(* LS Electric XG5000 project: XMC_MultiAxis_FBs *)
(* sample programs for multi-axis function blocks. *)
(* PLC LSPLC *)
(* module base 0 slot 0: Input/Output Module:XMC-DN24 (DC 24V Input 8Points/TR output 16Points) *)
(* module base 0 slot 1: Internal Analog Input/Output:XMF-AH04E (A/D voltage/current 2 channels, D/A voltage 2 channels) *)
(* task Periodic Task: Kind=2 *)
(* task Initialization Task: Kind=1 *)
(* task NC Program: Kind=6 *)

PROGRAM ECAT_Connect_Example (* task: Scan Program *)
VAR
    Connect_Error : BOOL; (* status that LS_Connect has an error *)
    Connect_ErrorID : WORD; (* LS_Connect Error number *)
    Connect_INST : LS_CONNECT; (* LS_Connect fb *)
    Disconnect_Error : BOOL; (* status that LS_Disconnect has an error *)
    Disconnect_ErrorID : WORD; (* Error Number for LS_Disconnect FB *)
    Disconnect_INST : LS_DISCONNECT; (* LS_Disconnect fb *)
    Execute_Connect : BOOL; (* Execute LS_Connect fb *)
    Execute_Disconnect : BOOL; (* execute LS_Disconnect fb *)
END_VAR

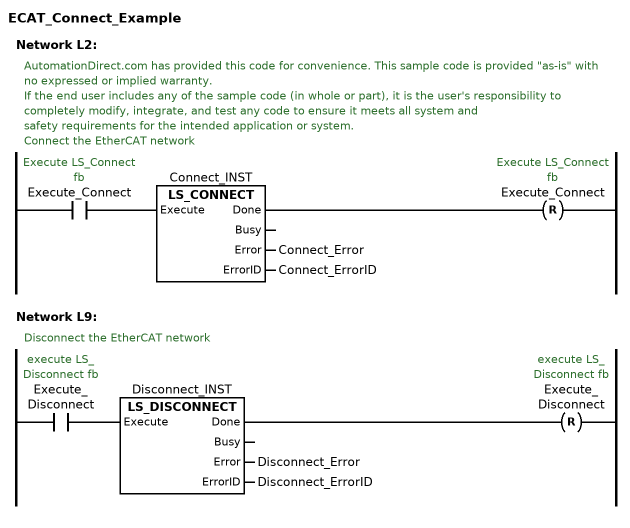
(* AutomationDirect.com has provided this code for convenience. This sample code is provided "as-is" with no expressed or implied warranty. / If the end user includes any of the sample code (in whole or part), it is the user's responsibility to completely modify, integrate, and test any code to ensure it meets all system and / safety requirements for the intended application or system. *)
(* Connect the EtherCAT network *)
(* Rung L2 *)
Connect_INST(Execute := Execute_Connect, Error => Connect_Error, ErrorID => Connect_ErrorID);
IF Connect_INST.Done THEN Execute_Connect := FALSE; END_IF;
(* Disconnect the EtherCAT network *)
(* Rung L9 *)
Disconnect_INST(Execute := Execute_Disconnect, Error => Disconnect_Error, ErrorID => Disconnect_ErrorID);
IF Disconnect_INST.Done THEN Execute_Disconnect := FALSE; END_IF;
END_PROGRAM

PROGRAM MC_PowerAll_Example (* task: Scan Program *)
(* example program for MC_PowerAll *)
VAR
    All_Axes_Ready : BOOL; (* flag that all axes are ready *)
    PowerAll_Error : BOOL; (* status of MC_Power error status *)
    PowerAll_ErrorID : WORD; (* error id of Axis 1 MC_Power *)
    PowerAll_INST : MC_POWERALL; (* MC_PowerALL fb *)
    PowerAll_Status : BOOL; (* status of axis 1 power *)
    PowerAll_Valid : BOOL; (* Axis1 power status is valid *)
    Power_On_Axis1 : BOOL; (* command to turn on power to axis 1 *)
END_VAR

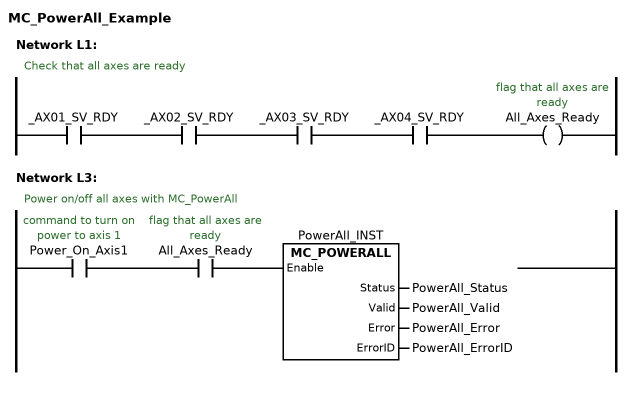
(* Check that all axes are ready *)
(* Rung L1 *)
All_Axes_Ready := _AX01_SV_RDY AND _AX02_SV_RDY AND _AX03_SV_RDY AND _AX04_SV_RDY;
(* Power on/off all axes with MC_PowerAll *)
(* Rung L3 *)
PowerAll_INST(Enable := Power_On_Axis1 AND All_Axes_Ready, Status => PowerAll_Status, Valid => PowerAll_Valid, Error => PowerAll_Error, ErrorID => PowerAll_ErrorID);
END_PROGRAM

PROGRAM Home_Example (* task: Scan Program *)
(* example of MC_Home and LS_Home *)
VAR
    All_Axes_Pwr_On : BOOL; (* status that all axes are powered on *)
    All_Axes_Ready : BOOL; (* flag that all axes are ready *)
    Execute_LS_HomeAll : BOOL; (* Execute LS_Home fb *)
    Execute_MC_HomeAll : BOOL; (* execute MC_Home fb *)
    LSHomeAll_Aborted : BOOL; (* LS_Home fb command aborted status *)
    LSHomeAll_Active : BOOL; (* LS_Home fb active status *)
    LSHomeAll_Busy : BOOL; (* LS_Home busy status *)
    LSHomeAll_Error : BOOL; (* LSHome fb error status *)
    LSHomeAll_ErrorID : WORD; (* LS_Home fb error id value *)
    LSHomeAll_INST : LS_HOMEALL; (* LS_HomeAll fb *)
    MCHomeAll_Aborted : BOOL; (* MC_Home command was aborted *)
    MCHomeAll_Active : BOOL; (* MC_Home is active *)
    MCHomeAll_Busy : BOOL; (* MC_Home is busy *)
    MCHomeAll_Error : BOOL; (* error status of MC_Home *)
    MCHomeAll_ErrorID : WORD; (* error id value for MC_Home *)
    MCHomeAll_INST : MC_HOMEALL; (* MC_HomeAll fb *)
END_VAR

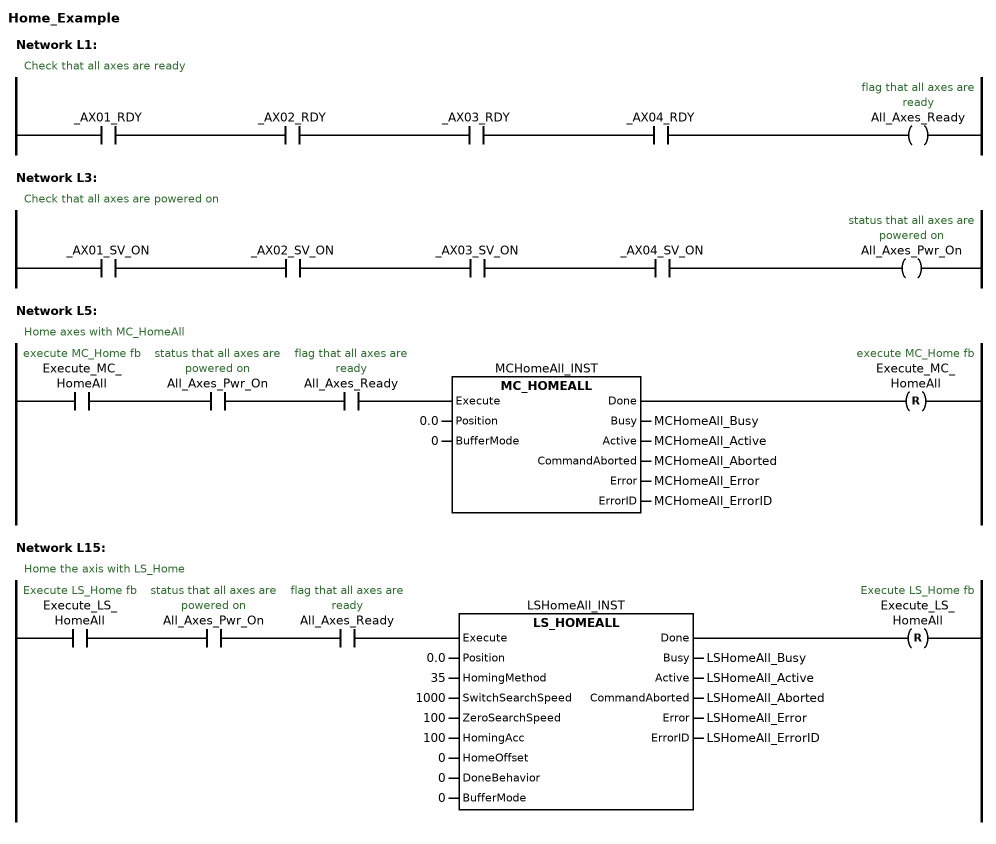
(* Check that all axes are ready *)
(* Rung L1 *)
All_Axes_Ready := _AX01_RDY AND _AX02_RDY AND _AX03_RDY AND _AX04_RDY;
(* Check that all axes are powered on *)
(* Rung L3 *)
All_Axes_Pwr_On := _AX01_SV_ON AND _AX02_SV_ON AND _AX03_SV_ON AND _AX04_SV_ON;
(* Home axes with MC_HomeAll *)
(* Rung L5 *)
MCHomeAll_INST(Execute := Execute_MC_HomeAll AND All_Axes_Pwr_On AND All_Axes_Ready, Position := 0.0, BufferMode := 0, Busy => MCHomeAll_Busy, Active => MCHomeAll_Active, CommandAborted => MCHomeAll_Aborted, Error => MCHomeAll_Error, ErrorID => MCHomeAll_ErrorID);
IF MCHomeAll_INST.Done THEN Execute_MC_HomeAll := FALSE; END_IF;
(* Home the axis with LS_Home *)
(* Rung L15 *)
LSHomeAll_INST(Execute := Execute_LS_HomeAll AND All_Axes_Pwr_On AND All_Axes_Ready, Position := 0.0, HomingMethod := 35, SwitchSearchSpeed := 1000, ZeroSearchSpeed := 100, HomingAcc := 100, HomeOffset := 0, DoneBehavior := 0, BufferMode := 0, Busy => LSHomeAll_Busy, Active => LSHomeAll_Active, CommandAborted => LSHomeAll_Aborted, Error => LSHomeAll_Error, ErrorID => LSHomeAll_ErrorID);
IF LSHomeAll_INST.Done THEN Execute_LS_HomeAll := FALSE; END_IF;
END_PROGRAM

PROGRAM MCStopAll_MCHaltAll_Examples (* task: Scan Program *)
(* Examples of MC_Stop and MC_Hault function blocks. *)
VAR
    All_Axes_Pwr_On : BOOL; (* status that all axes are powered on *)
    All_Axes_Ready : BOOL; (* flag that all axes are ready *)
    Execute_MCHaltAll : BOOL; (* execute MC_Halt FB *)
    Execute_MCStopAll : BOOL; (* command to execute MC_Stop fb *)
    MCHaltAll_Aborted : BOOL; (* MC_Hault command aborted status *)
    MCHaltAll_Active : BOOL; (* MC_Halt active status *)
    MCHaltAll_Busy : BOOL; (* Busy status for MC_Halt *)
    MCHaltAll_Error : BOOL; (* MC_Halt error status *)
    MCHaltAll_ErrorID : WORD; (* MC_Halt Error identification value *)
    MCHaltAll_INST : MC_HALTALL; (* MC_HaltAll fb *)
    MCStopAll_Aborted : BOOL; (* MC_Stop aborted status *)
    MCStopAll_Busy : BOOL; (* MC_Stop Busy Status *)
    MCStopAll_Error : BOOL; (* MC_Stop error status *)
    MCStopAll_ErrorID : WORD; (* MC_Stop error identification value *)
    MCStopAll_INST : MC_STOPALL; (* MC_Stop function block *)
END_VAR

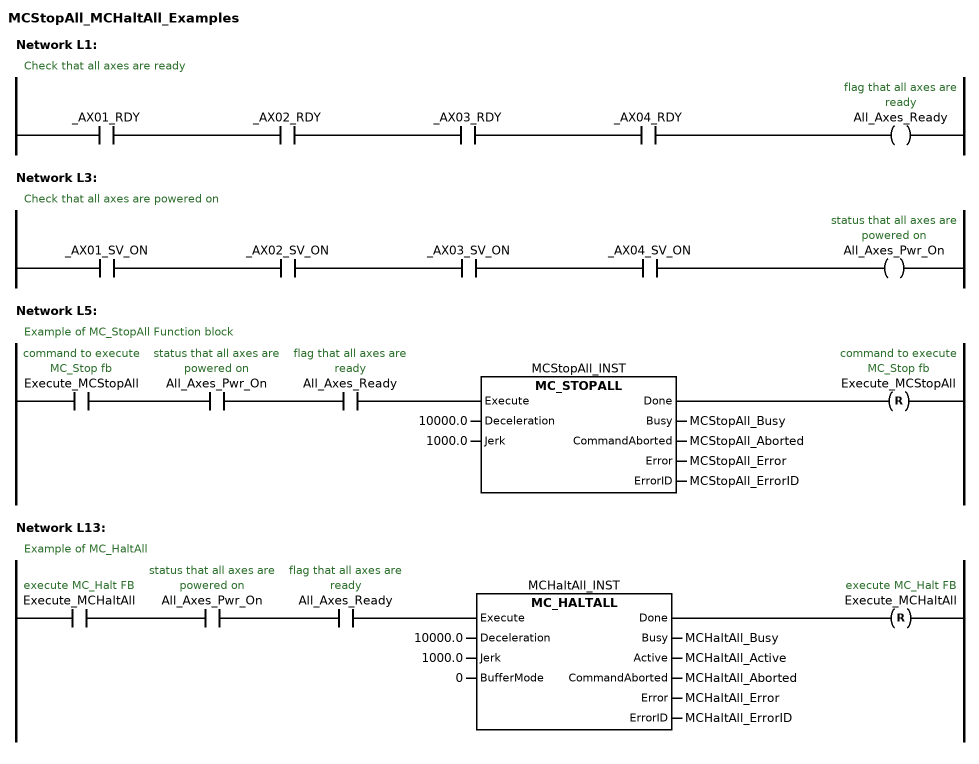
(* Check that all axes are ready *)
(* Rung L1 *)
All_Axes_Ready := _AX01_RDY AND _AX02_RDY AND _AX03_RDY AND _AX04_RDY;
(* Check that all axes are powered on *)
(* Rung L3 *)
All_Axes_Pwr_On := _AX01_SV_ON AND _AX02_SV_ON AND _AX03_SV_ON AND _AX04_SV_ON;
(* Example of MC_StopAll Function block *)
(* Rung L5 *)
MCStopAll_INST(Execute := Execute_MCStopAll AND All_Axes_Pwr_On AND All_Axes_Ready, Deceleration := 10000.0, Jerk := 1000.0, Busy => MCStopAll_Busy, CommandAborted => MCStopAll_Aborted, Error => MCStopAll_Error, ErrorID => MCStopAll_ErrorID);
IF MCStopAll_INST.Done THEN Execute_MCStopAll := FALSE; END_IF;
(* Example of MC_HaltAll *)
(* Rung L13 *)
MCHaltAll_INST(Execute := Execute_MCHaltAll AND All_Axes_Pwr_On AND All_Axes_Ready, Deceleration := 10000.0, Jerk := 1000.0, BufferMode := 0, Busy => MCHaltAll_Busy, Active => MCHaltAll_Active, CommandAborted => MCHaltAll_Aborted, Error => MCHaltAll_Error, ErrorID => MCHaltAll_ErrorID);
IF MCHaltAll_INST.Done THEN Execute_MCHaltAll := FALSE; END_IF;
END_PROGRAM

PROGRAM MC_Reset2All_Example (* task: Scan Program *)
(* example of MC_Reset2All function block. *)
VAR
    All_Axes_Ready : BOOL; (* flag that all axes are ready *)
    Execute_MCReset2All : BOOL; (* command to execute MC_Reset2 *)
    Reset2All_Busy : BOOL; (* busy status for MC_Reset2 *)
    Reset2All_Error : BOOL; (* error status for MC_Reset2 *)
    Reset2All_ErrorID : WORD; (* MC_Reset2 error identification *)
    Reset2All_ErrorType : UINT; (* error type for MC_Reset2 *)
    Reset2All_INST : MC_RESET2ALL; (* MC_Reset2All fb *)
END_VAR

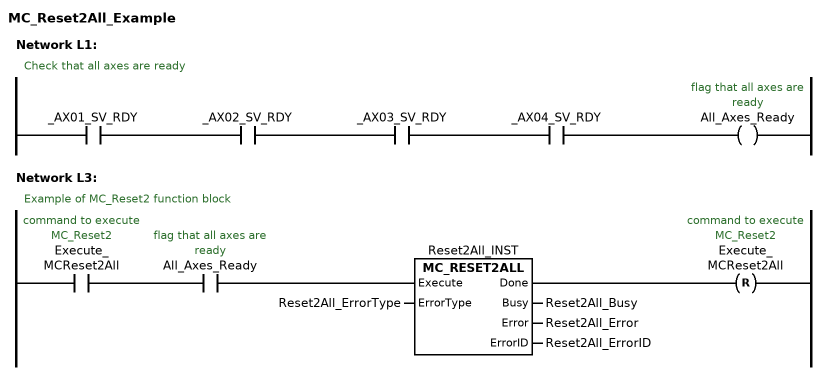
(* Check that all axes are ready *)
(* Rung L1 *)
All_Axes_Ready := _AX01_SV_RDY AND _AX02_SV_RDY AND _AX03_SV_RDY AND _AX04_SV_RDY;
(* Example of MC_Reset2 function block *)
(* Rung L3 *)
Reset2All_INST(Execute := Execute_MCReset2All AND All_Axes_Ready, ErrorType := Reset2All_ErrorType, Busy => Reset2All_Busy, Error => Reset2All_Error, ErrorID => Reset2All_ErrorID);
IF Reset2All_INST.Done THEN Execute_MCReset2All := FALSE; END_IF;
END_PROGRAM

PROGRAM MC_CamIn_CamOut_Example (* task: Scan Program *)
(* Example of MC_CamIn and MC_CamOut function block *)
VAR
    All_Axes_Pwr_On : BOOL; (* status that all axes are powered on *)
    All_Axes_Ready : BOOL; (* flag that all axes are ready *)
    CamIn_Aborted : BOOL; (* MC_CamIn command aborted status *)
    CamIn_Active : BOOL; (* MC_CamIn active status *)
    CamIn_Busy : BOOL; (* MC_CamIn busy status *)
    CamIn_CamTableID : UINT; (* Cam profle table id for MC_CamIn *)
    CamIn_ContinuousUpdate : BOOL; (* Continuous update input of MC_CamIn *)
    CamIn_EndOfProfile : BOOL; (* MC_CamIn end of profile status *)
    CamIn_Error : BOOL; (* MC_CamIn error status *)
    CamIn_ErrorID : WORD; (* MC_CamIn error identification *)
    CamIn_INST : MC_CAMIN; (* MC_CamIn fb *)
    CamIn_MasterOffset : LREAL; (* Master offset of MC_CamIn *)
    CamIn_MasterScaling : LREAL; (* Master scaling for MC_CamIn *)
    CamIn_MasterStartDistance : LREAL; (* Master Start distance for MC_CamIn *)
    CamIn_MasterSyncPosition : LREAL; (* Master Sync Position for MC_CamIn *)
    CamIn_MasterValueSource : UINT; (* Master value source for MC_CamIn *)
    CamIn_SlaveOffset : LREAL; (* Slave offset of MC_CamIn *)
    CamIn_SlaveScaling : LREAL; (* slave scaling MC_CamIn *)
    CamIn_StartMode : UINT; (* Start mode for MC_CamIn *)
    CamOut_Busy : BOOL; (* MC_CamOut busy status *)
    CamOut_Error : BOOL; (* error status for MC_CamOut *)
    CamOut_ErrorID : WORD; (* Error identification for MC_CamOut *)
    CamOut_INST : MC_CAMOUT; (* MC_CamOut function block *)
    Execute_CamIn : BOOL; (* execute MC_CamIn *)
    Execute_CamOut : BOOL; (* execute MC_CamOut function block *)
    Execute_MoveVelocity : BOOL; (* execute the MC_MoveVelocity Function block *)
    Master_Axis : UINT; (* master axis of MC_CamIn *)
    Slave_Axis : UINT; (* slave axis of MC_CamIn *)
    VelocityMove_Aborted : BOOL; (* MC_MoveVelocity Status aborted *)
    VelocityMove_Active : BOOL; (* active status of MC_MoveVelocity *)
    VelocityMove_Busy : BOOL; (* busy status of MC_MoveVelocity *)
    VelocityMove_Error : BOOL; (* Error status of MC_MoveVelocity *)
    VelocityMove_ErrorID : WORD; (* MC_MoveVelocity error identification *)
    Velocity_INST : MC_MOVEVELOCITY; (* MC_MoveVelocity function block instance *)
END_VAR

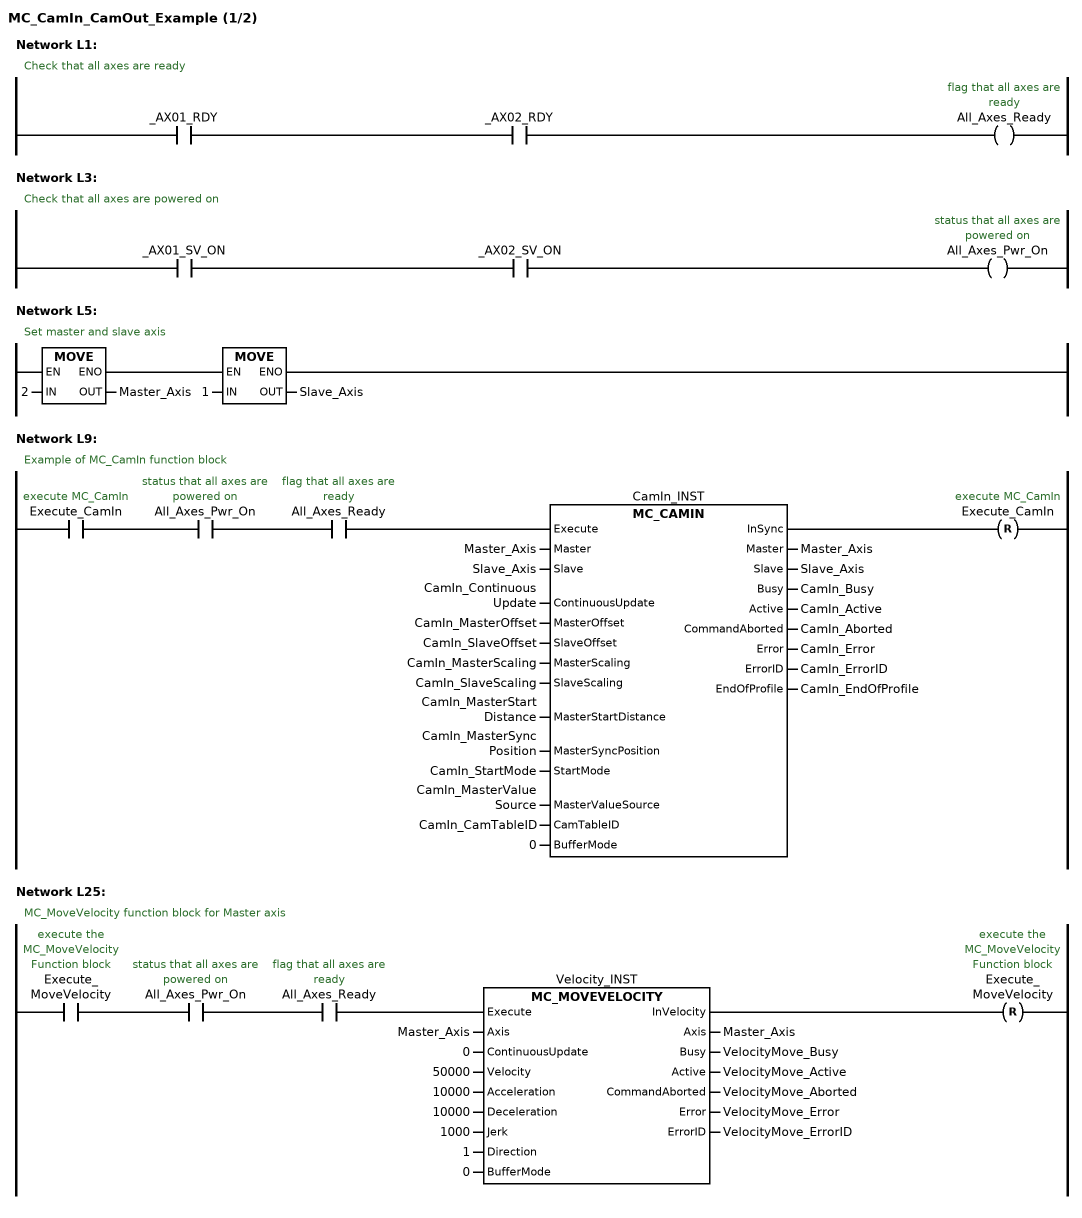
(* Check that all axes are ready *)
(* Rung L1 *)
All_Axes_Ready := _AX01_RDY AND _AX02_RDY;
(* Check that all axes are powered on *)
(* Rung L3 *)
All_Axes_Pwr_On := _AX01_SV_ON AND _AX02_SV_ON;
(* Set master and slave axis *)
(* Rung L5 *)
Master_Axis := 2;
Slave_Axis := 1;
(* Example of MC_CamIn function block *)
(* Rung L9 *)
CamIn_INST(Execute := Execute_CamIn AND All_Axes_Pwr_On AND All_Axes_Ready, Master := Master_Axis, Slave := Slave_Axis, ContinuousUpdate := CamIn_ContinuousUpdate, MasterOffset := CamIn_MasterOffset, SlaveOffset := CamIn_SlaveOffset, MasterScaling := CamIn_MasterScaling, SlaveScaling := CamIn_SlaveScaling, MasterStartDistance := CamIn_MasterStartDistance, MasterSyncPosition := CamIn_MasterSyncPosition, StartMode := CamIn_StartMode, MasterValueSource := CamIn_MasterValueSource, CamTableID := CamIn_CamTableID, BufferMode := 0, Master => Master_Axis, Slave => Slave_Axis, Busy => CamIn_Busy, Active => CamIn_Active, CommandAborted => CamIn_Aborted, Error => CamIn_Error, ErrorID => CamIn_ErrorID, EndOfProfile => CamIn_EndOfProfile);
IF CamIn_INST.InSync THEN Execute_CamIn := FALSE; END_IF;
(* MC_MoveVelocity function block for Master axis *)
(* Rung L25 *)
Velocity_INST(Execute := Execute_MoveVelocity AND All_Axes_Pwr_On AND All_Axes_Ready, Axis := Master_Axis, ContinuousUpdate := 0, Velocity := 50000, Acceleration := 10000, Deceleration := 10000, Jerk := 1000, Direction := 1, BufferMode := 0, Axis => Master_Axis, Busy => VelocityMove_Busy, Active => VelocityMove_Active, CommandAborted => VelocityMove_Aborted, Error => VelocityMove_Error, ErrorID => VelocityMove_ErrorID);
IF Velocity_INST.InVelocity THEN Execute_MoveVelocity := FALSE; END_IF;

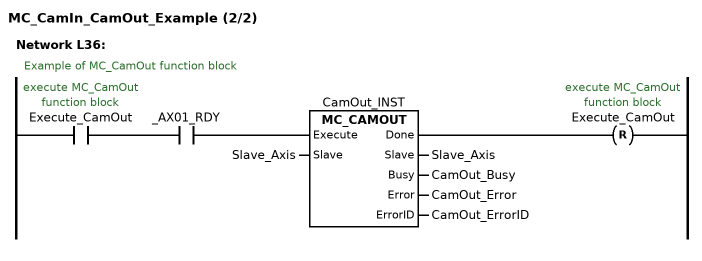
(* Example of MC_CamOut function block *)
(* Rung L36 *)
CamOut_INST(Execute := Execute_CamOut AND _AX01_RDY, Slave := Slave_Axis, Slave => Slave_Axis, Busy => CamOut_Busy, Error => CamOut_Error, ErrorID => CamOut_ErrorID);
IF CamOut_INST.Done THEN Execute_CamOut := FALSE; END_IF;
END_PROGRAM

PROGRAM MC_GearIn_GearInEx_GearOut_Example (* task: Scan Program *)
(* example of MC_GearIn and MC_GearOut function blocks *)
VAR
    All_Axes_Pwr_On : BOOL; (* status that all axes are powered on *)
    All_Axes_Ready : BOOL; (* flag that all axes are ready *)
    Execute_GearIn : BOOL; (* execute MC_GearIn fb *)
    Execute_GearInEx : BOOL; (* execute MC_GearInEx function block *)
    Execute_GearOut : BOOL; (* execute MC_GearOut fb *)
    Execute_MoveVelocity : BOOL; (* execute the MC_MoveVelocity Function block *)
    GearInEx_Aborted : BOOL; (* aborted status for MC_GearInEx *)
    GearInEx_Acceleration : LREAL; (* accleration for MC_GearInEx *)
    GearInEx_Active : BOOL; (* active status for MC_GearInEx *)
    GearInEx_Busy : BOOL; (* busy status for MC_GearInEx *)
    GearInEx_ContinuousUpdate : BOOL; (* continuous update for MC_GearInEx *)
    GearInEx_Deceleration : LREAL; (* deceleration for MC_GearInEx *)
    GearInEx_Error : BOOL; (* error status for MC_GearInEx *)
    GearInEx_ErrorID : WORD; (* error identification for MC_GearInEx *)
    GearInEx_INST : MC_GEARINEX; (* MC_GearInEx function block *)
    GearInEx_Jerk : LREAL; (* jerk value for MC_GearInEx *)
    GearInEx_MasterValueSource : UINT; (* MasterValueSource for MC_GearInEx *)
    GearInEx_RatioDenominator : UDINT; (* ratio denominator for MC_GearInEx *)
    GearInEx_RatioNumerator : DINT; (* ratio numerator for MC_GearInEx *)
    GearIn_Aborted : BOOL; (* aborted status for MC_GearIn *)
    GearIn_Acceleration : LREAL; (* Acceleration for MC_GearIn *)
    GearIn_Active : BOOL; (* active status for MC_GearIn *)
    GearIn_Busy : BOOL; (* busy value for MC_GearIn *)
    GearIn_ContinuousUpdate : BOOL; (* Continuous Update of MC_GearIn *)
    GearIn_Deceleration : LREAL; (* Deceleration for MC_GearIn *)
    GearIn_Error : BOOL; (* error status for MC_GearIn *)
    GearIn_ErrorID : WORD; (* error identification for MC_GearIn *)
    GearIn_INST : MC_GEARIN; (* MC_GearIn fb *)
    GearIn_Jerk : LREAL; (* Jerk value for MC_GearIn *)
    GearIn_MasterValueSource : UINT; (* choose commanded or current position from master *)
    GearIn_RatioDenominator : UINT; (* Denominator for MC_GearIn *)
    GearIn_RatioNumerator : INT; (* Numerator for MC_Gearin *)
    GearOut_Busy : BOOL; (* busy status of MC_GearOut *)
    GearOut_Error : BOOL; (* error status of MC_GearOut *)
    GearOut_ErrorID : WORD; (* error identification of MC_GearOut *)
    GearOut_INST : MC_GEAROUT; (* MC_GearOut fb *)
    Master_Axis : UINT; (* master axis of MC_CamIn *)
    Slave_Axis : UINT; (* slave axis of MC_CamIn *)
    VelocityMove_Aborted : BOOL; (* MC_MoveVelocity Status aborted *)
    VelocityMove_Active : BOOL; (* active status of MC_MoveVelocity *)
    VelocityMove_Busy : BOOL; (* busy status of MC_MoveVelocity *)
    VelocityMove_Error : BOOL; (* Error status of MC_MoveVelocity *)
    VelocityMove_ErrorID : WORD; (* MC_MoveVelocity error identification *)
    Velocity_INST : MC_MOVEVELOCITY; (* MC_MoveVelocity function block instance *)
END_VAR

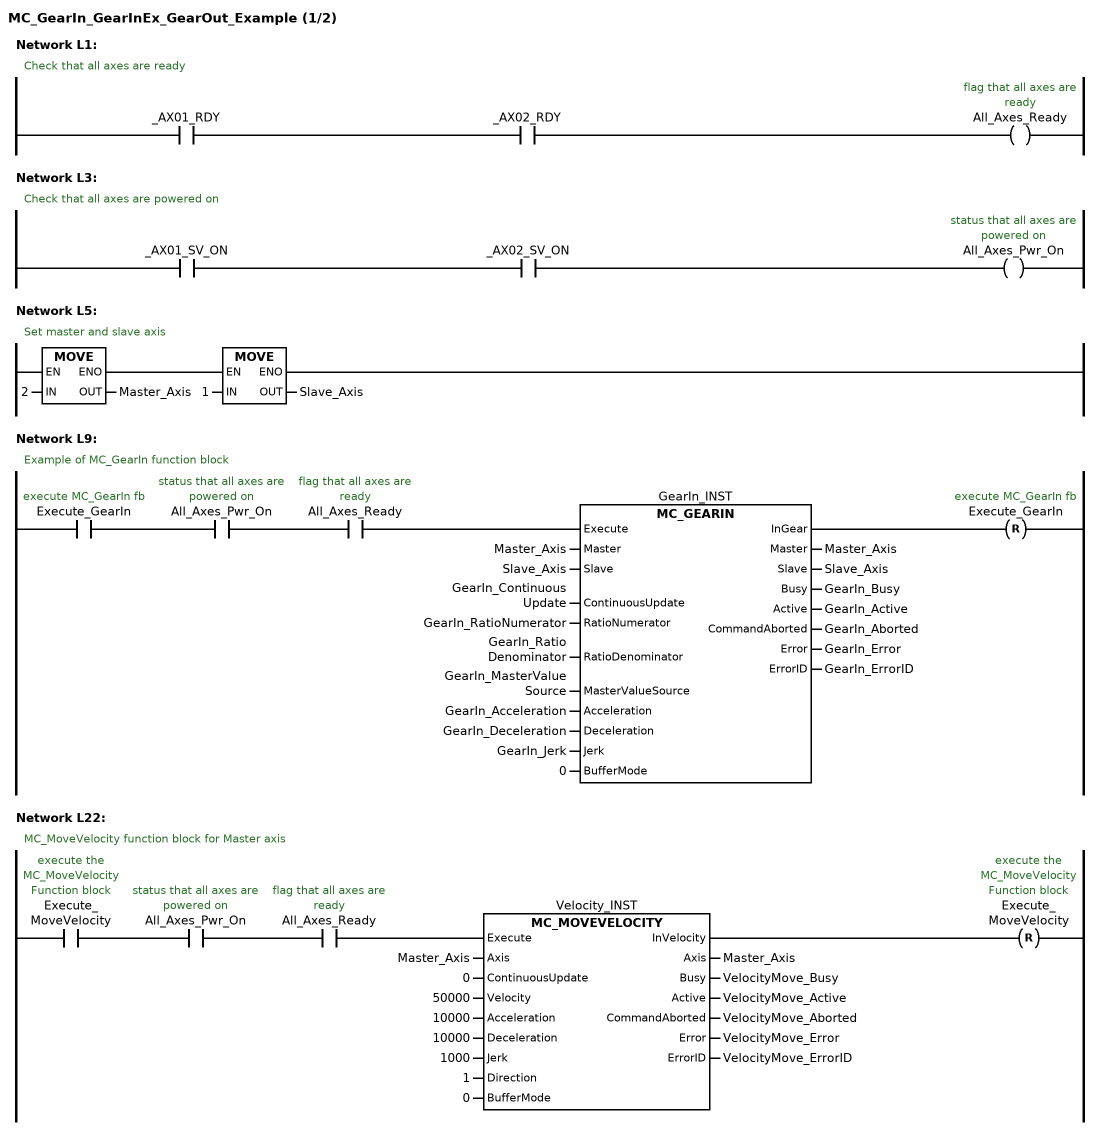
(* Check that all axes are ready *)
(* Rung L1 *)
All_Axes_Ready := _AX01_RDY AND _AX02_RDY;
(* Check that all axes are powered on *)
(* Rung L3 *)
All_Axes_Pwr_On := _AX01_SV_ON AND _AX02_SV_ON;
(* Set master and slave axis *)
(* Rung L5 *)
Master_Axis := 2;
Slave_Axis := 1;
(* Example of MC_GearIn function block *)
(* Rung L9 *)
GearIn_INST(Execute := Execute_GearIn AND All_Axes_Pwr_On AND All_Axes_Ready, Master := Master_Axis, Slave := Slave_Axis, ContinuousUpdate := GearIn_ContinuousUpdate, RatioNumerator := GearIn_RatioNumerator, RatioDenominator := GearIn_RatioDenominator, MasterValueSource := GearIn_MasterValueSource, Acceleration := GearIn_Acceleration, Deceleration := GearIn_Deceleration, Jerk := GearIn_Jerk, BufferMode := 0, Master => Master_Axis, Slave => Slave_Axis, Busy => GearIn_Busy, Active => GearIn_Active, CommandAborted => GearIn_Aborted, Error => GearIn_Error, ErrorID => GearIn_ErrorID);
IF GearIn_INST.InGear THEN Execute_GearIn := FALSE; END_IF;
(* MC_MoveVelocity function block for Master axis *)
(* Rung L22 *)
Velocity_INST(Execute := Execute_MoveVelocity AND All_Axes_Pwr_On AND All_Axes_Ready, Axis := Master_Axis, ContinuousUpdate := 0, Velocity := 50000, Acceleration := 10000, Deceleration := 10000, Jerk := 1000, Direction := 1, BufferMode := 0, Axis => Master_Axis, Busy => VelocityMove_Busy, Active => VelocityMove_Active, CommandAborted => VelocityMove_Aborted, Error => VelocityMove_Error, ErrorID => VelocityMove_ErrorID);
IF Velocity_INST.InVelocity THEN Execute_MoveVelocity := FALSE; END_IF;

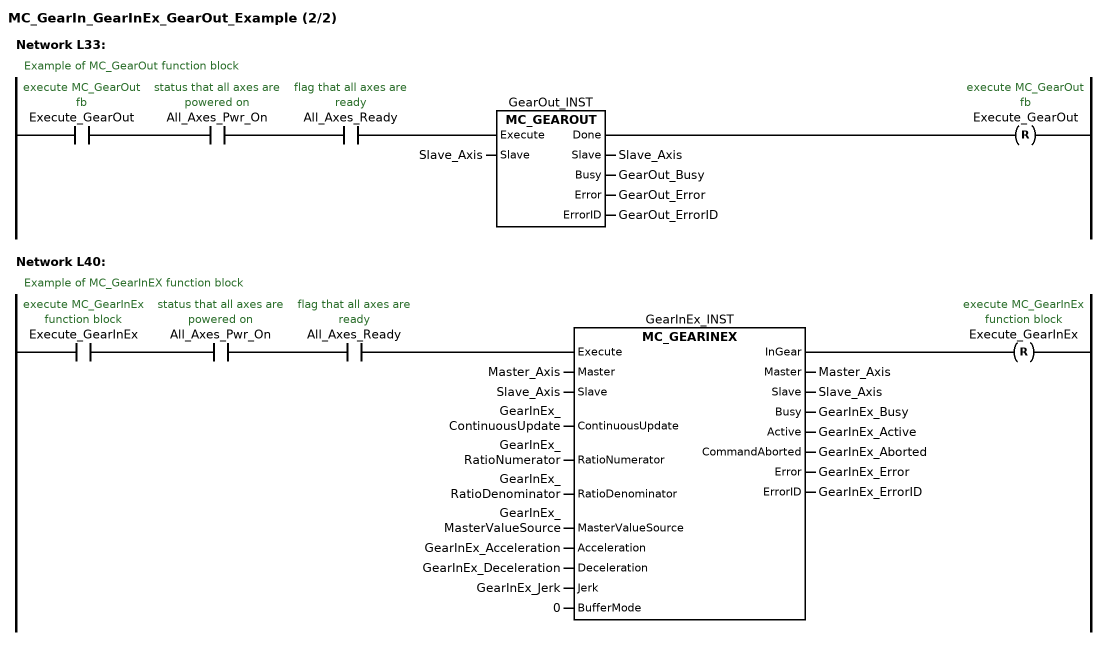
(* Example of MC_GearOut function block *)
(* Rung L33 *)
GearOut_INST(Execute := Execute_GearOut AND All_Axes_Pwr_On AND All_Axes_Ready, Slave := Slave_Axis, Slave => Slave_Axis, Busy => GearOut_Busy, Error => GearOut_Error, ErrorID => GearOut_ErrorID);
IF GearOut_INST.Done THEN Execute_GearOut := FALSE; END_IF;
(* Example of MC_GearInEX function block *)
(* Rung L40 *)
GearInEx_INST(Execute := Execute_GearInEx AND All_Axes_Pwr_On AND All_Axes_Ready, Master := Master_Axis, Slave := Slave_Axis, ContinuousUpdate := GearInEx_ContinuousUpdate, RatioNumerator := GearInEx_RatioNumerator, RatioDenominator := GearInEx_RatioDenominator, MasterValueSource := GearInEx_MasterValueSource, Acceleration := GearInEx_Acceleration, Deceleration := GearInEx_Deceleration, Jerk := GearInEx_Jerk, BufferMode := 0, Master => Master_Axis, Slave => Slave_Axis, Busy => GearInEx_Busy, Active => GearInEx_Active, CommandAborted => GearInEx_Aborted, Error => GearInEx_Error, ErrorID => GearInEx_ErrorID);
IF GearInEx_INST.InGear THEN Execute_GearInEx := FALSE; END_IF;
END_PROGRAM

PROGRAM MC_GearInPos_GearInPosEX_Example (* task: Scan Program *)
(* exmple program for MC_GearInPos and MC_GearInPosEx function blocks *)
VAR
    All_Axes_Pwr_On : BOOL; (* status that all axes are powered on *)
    All_Axes_Ready : BOOL; (* flag that all axes are ready *)
    Execute_GearInPos : BOOL; (* execute MC_GearInPos function block *)
    Execute_GearInPosEx : BOOL; (* execute MC_GearInPosEx function block *)
    Execute_MoveRelative : BOOL; (* execute the MC_MoveVelocity Function block *)
    GearInPosEx_Aborted : BOOL; (* command aborted status for MC_GearInPosEx *)
    GearInPosEx_Acceleration : LREAL; (* acceleration for MC_GearInPosEx *)
    GearInPosEx_Active : BOOL; (* active status for MC_GearInPosEx *)
    GearInPosEx_Busy : BOOL; (* busy status for MC_GearInPosEx *)
    GearInPosEx_Deceleration : LREAL; (* deceleration for MC_GearInPosEx *)
    GearInPosEx_Error : BOOL; (* error status for MC_GearInPosEx *)
    GearInPosEx_ErrorID : WORD; (* error identification for MC_GearInPosEx *)
    GearInPosEx_INST : MC_GEARINPOSEX; (* MC_GearInPosEx function block *)
    GearInPosEx_Jerk : LREAL; (* jerk for MC_GearInPosEx *)
    GearInPosEx_MasterStartDistance : LREAL; (* Master Start Distance for MC_GearInPosEx *)
    GearInPosEx_MasterSyncPosition : LREAL; (* Master sync position for MC_GearInPosEx *)
    GearInPosEx_MasterValueSource : UINT; (* MasterValueSource for MC_GearInPosEx *)
    GearInPosEx_RatioDenominator : UDINT; (* ratio denominator for MC_GearInPosEx *)
    GearInPosEx_RatioNumerator : DINT; (* Ratio numerator for MC_GearInPosEx *)
    GearInPosEx_SlaveSyncPosition : LREAL; (* Slave Sync Position for MC_GearInPosEx *)
    GearInPosEx_StartSync : BOOL; (* start sync status for MC_GearInPosEx *)
    GearInPosEx_Velocity : LREAL; (* Velocity for MC_GearInPosEx *)
    GearInPos_Aborted : BOOL; (* aborted status for MC_GearInPos *)
    GearInPos_Acceleration : LREAL; (* Acceleration for MC_GearInPos *)
    GearInPos_Active : BOOL; (* active status for MC_GearInPos *)
    GearInPos_Busy : BOOL; (* busy status for MC_GearInPos *)
    GearInPos_Deceleration : LREAL; (* Deceleration for MC_GearInPos *)
    GearInPos_Error : BOOL; (* error status for MC_GearInPos *)
    GearInPos_ErrorID : WORD; (* error identification for MC_GearInPos *)
    GearInPos_INST : MC_GEARINPOS; (* MC_GearInPos function block *)
    GearInPos_Jerk : LREAL; (* Jerk value for MC_GearInPos *)
    GearInPos_MasterStartDistance : LREAL; (* MasterStartDistance for MC_GearInPos *)
    GearInPos_MasterSyncPosition : LREAL; (* MasterSyncPosition for MC_GearInPos *)
    GearInPos_MasterValueSource : UINT; (* MasterValueSource for MC_GearInPos *)
    GearInPos_RatioDenominator : UINT; (* ratio denominator for MC_GearInPos *)
    GearInPos_RatioNumerator : INT; (* ratio numerator for MC_GearInPos *)
    GearInPos_SlaveSyncPosition : LREAL; (* SlaveSyncPosition for MC_GearInPos *)
    GearInPos_StartSync : BOOL; (* StartSync status for MC_GearInPos *)
    GearInPos_Velocity : LREAL; (* Velocity for MC_GearInPos *)
    Master_Axis : UINT; (* master axis of MC_CamIn *)
    MoveRelative_INST : MC_MOVERELATIVE;
    Slave_Axis : UINT; (* slave axis of MC_CamIn *)
END_VAR

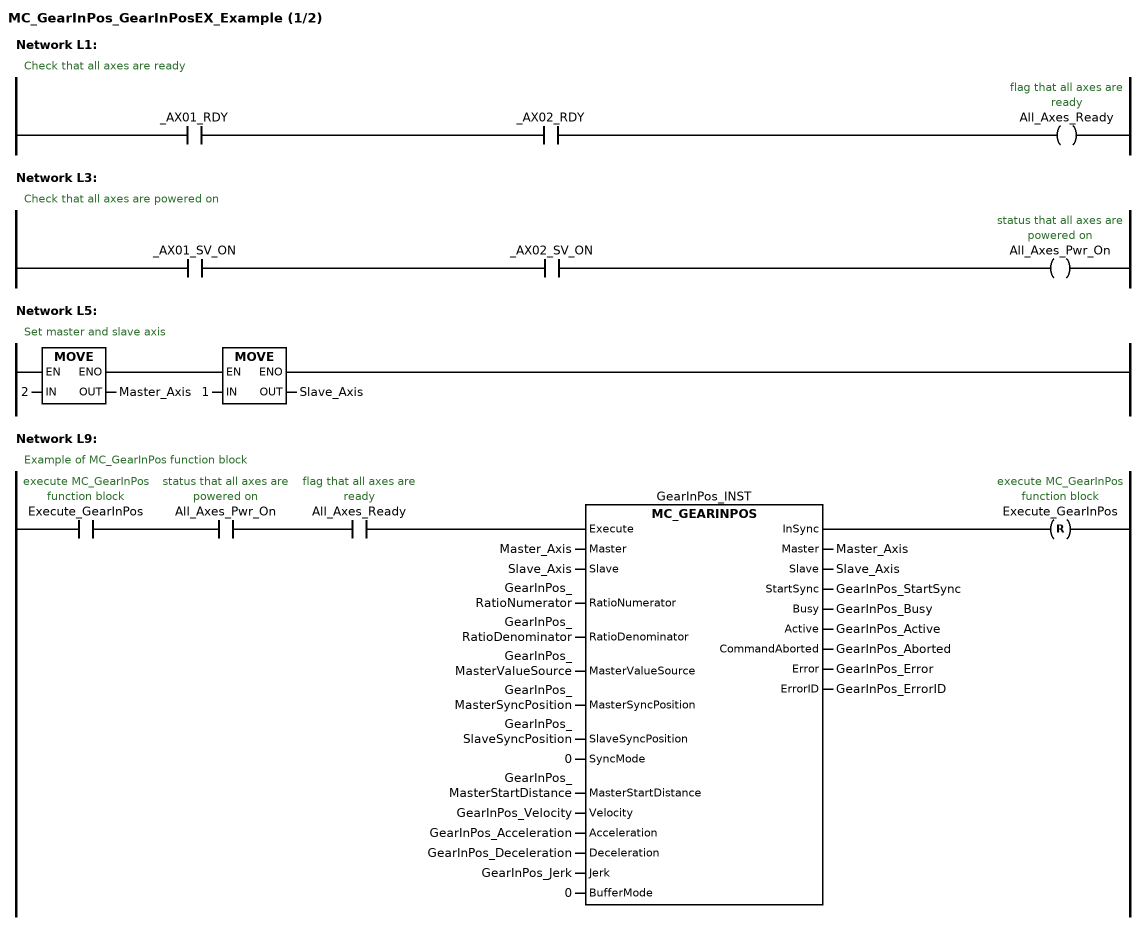
(* Check that all axes are ready *)
(* Rung L1 *)
All_Axes_Ready := _AX01_RDY AND _AX02_RDY;
(* Check that all axes are powered on *)
(* Rung L3 *)
All_Axes_Pwr_On := _AX01_SV_ON AND _AX02_SV_ON;
(* Set master and slave axis *)
(* Rung L5 *)
Master_Axis := 2;
Slave_Axis := 1;
(* Example of MC_GearInPos function block *)
(* Rung L9 *)
GearInPos_INST(Execute := Execute_GearInPos AND All_Axes_Pwr_On AND All_Axes_Ready, Master := Master_Axis, Slave := Slave_Axis, RatioNumerator := GearInPos_RatioNumerator, RatioDenominator := GearInPos_RatioDenominator, MasterValueSource := GearInPos_MasterValueSource, MasterSyncPosition := GearInPos_MasterSyncPosition, SlaveSyncPosition := GearInPos_SlaveSyncPosition, SyncMode := 0, MasterStartDistance := GearInPos_MasterStartDistance, Velocity := GearInPos_Velocity, Acceleration := GearInPos_Acceleration, Deceleration := GearInPos_Deceleration, Jerk := GearInPos_Jerk, BufferMode := 0, Master => Master_Axis, Slave => Slave_Axis, StartSync => GearInPos_StartSync, Busy => GearInPos_Busy, Active => GearInPos_Active, CommandAborted => GearInPos_Aborted, Error => GearInPos_Error, ErrorID => GearInPos_ErrorID);
IF GearInPos_INST.InSync THEN Execute_GearInPos := FALSE; END_IF;

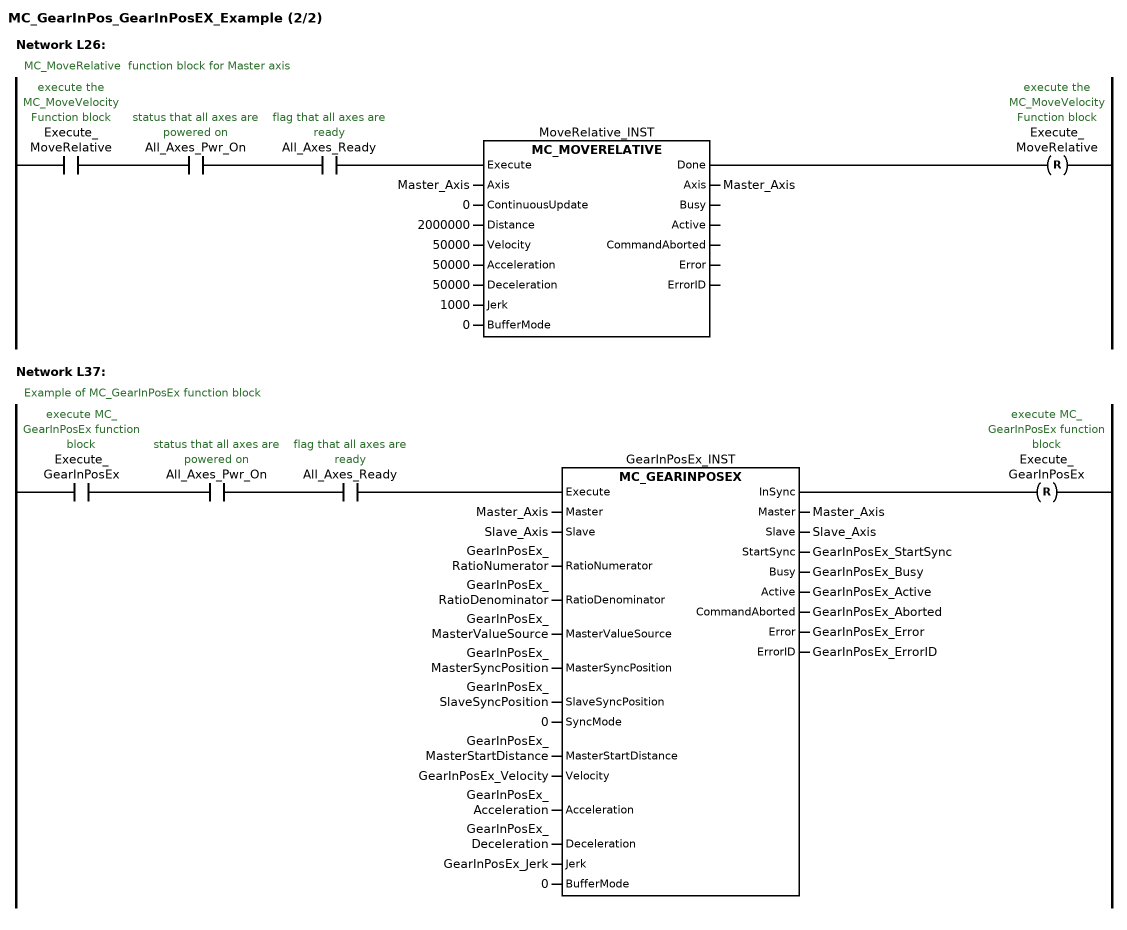
(* MC_MoveRelative  function block for Master axis *)
(* Rung L26 *)
MoveRelative_INST(Execute := Execute_MoveRelative AND All_Axes_Pwr_On AND All_Axes_Ready, Axis := Master_Axis, ContinuousUpdate := 0, Distance := 2000000, Velocity := 50000, Acceleration := 50000, Deceleration := 50000, Jerk := 1000, BufferMode := 0, Axis => Master_Axis);
IF MoveRelative_INST.Done THEN Execute_MoveRelative := FALSE; END_IF;
(* Example of MC_GearInPosEx function block *)
(* Rung L37 *)
GearInPosEx_INST(Execute := Execute_GearInPosEx AND All_Axes_Pwr_On AND All_Axes_Ready, Master := Master_Axis, Slave := Slave_Axis, RatioNumerator := GearInPosEx_RatioNumerator, RatioDenominator := GearInPosEx_RatioDenominator, MasterValueSource := GearInPosEx_MasterValueSource, MasterSyncPosition := GearInPosEx_MasterSyncPosition, SlaveSyncPosition := GearInPosEx_SlaveSyncPosition, SyncMode := 0, MasterStartDistance := GearInPosEx_MasterStartDistance, Velocity := GearInPosEx_Velocity, Acceleration := GearInPosEx_Acceleration, Deceleration := GearInPosEx_Deceleration, Jerk := GearInPosEx_Jerk, BufferMode := 0, Master => Master_Axis, Slave => Slave_Axis, StartSync => GearInPosEx_StartSync, Busy => GearInPosEx_Busy, Active => GearInPosEx_Active, CommandAborted => GearInPosEx_Aborted, Error => GearInPosEx_Error, ErrorID => GearInPosEx_ErrorID);
IF GearInPosEx_INST.InSync THEN Execute_GearInPosEx := FALSE; END_IF;
END_PROGRAM

PROGRAM MC_Phasing_Example (* task: Scan Program *)
(* Example program for MC_Phasing function block *)
VAR
    All_Axes_Pwr_On : BOOL; (* status that all axes are powered on *)
    All_Axes_Ready : BOOL; (* flag that all axes are ready *)
    Execute_Phasing : BOOL; (* execute MC_Phasing fb *)
    Master_Axis : UINT; (* master axis of MC_CamIn *)
    Phasing_Aborted : BOOL; (* aborted status for MC_Phasing *)
    Phasing_Acceleration : LREAL; (* acceleration for MC_Phasing *)
    Phasing_Active : BOOL; (* active status for MC_Phasing *)
    Phasing_Busy : BOOL; (* busy status for MC_Phasing *)
    Phasing_CoveredPhaseShift : LREAL; (* applied phase correction value for MC_Phasing *)
    Phasing_Deceleration : LREAL; (* deceleration for MC_Phasing *)
    Phasing_Error : BOOL; (* error status for MC_Phasing *)
    Phasing_ErrorID : WORD; (* error identification for MC_Phasing *)
    Phasing_INST : MC_PHASING; (* MC_Phasing FB *)
    Phasing_Jerk : LREAL; (* jerk value for MC_Phasing *)
    Phasing_PhaseShift : LREAL; (* phase compensation value *)
    Phasing_Velocity : LREAL; (* velocity for MC_Phasing *)
    Slave_Axis : UINT; (* slave axis of MC_CamIn *)
END_VAR

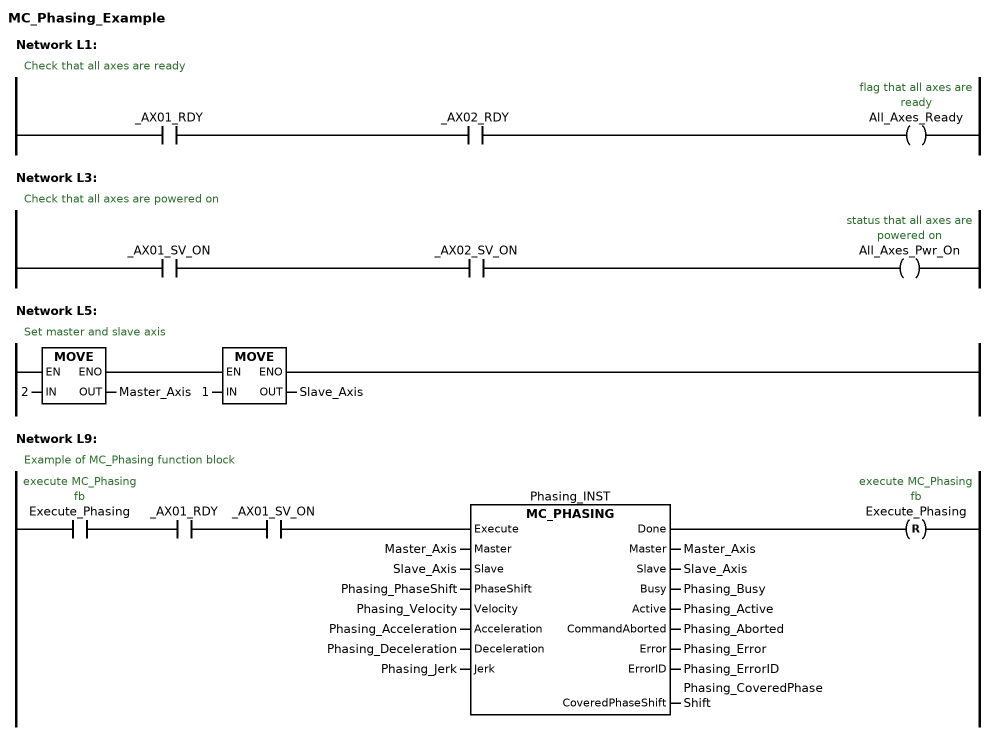
(* Check that all axes are ready *)
(* Rung L1 *)
All_Axes_Ready := _AX01_RDY AND _AX02_RDY;
(* Check that all axes are powered on *)
(* Rung L3 *)
All_Axes_Pwr_On := _AX01_SV_ON AND _AX02_SV_ON;
(* Set master and slave axis *)
(* Rung L5 *)
Master_Axis := 2;
Slave_Axis := 1;
(* Example of MC_Phasing function block *)
(* Rung L9 *)
Phasing_INST(Execute := Execute_Phasing AND _AX01_RDY AND _AX01_SV_ON, Master := Master_Axis, Slave := Slave_Axis, PhaseShift := Phasing_PhaseShift, Velocity := Phasing_Velocity, Acceleration := Phasing_Acceleration, Deceleration := Phasing_Deceleration, Jerk := Phasing_Jerk, Master => Master_Axis, Slave => Slave_Axis, Busy => Phasing_Busy, Active => Phasing_Active, CommandAborted => Phasing_Aborted, Error => Phasing_Error, ErrorID => Phasing_ErrorID, CoveredPhaseShift => Phasing_CoveredPhaseShift);
IF Phasing_INST.Done THEN Execute_Phasing := FALSE; END_IF;
END_PROGRAM

PROGRAM MC_SetPositionAll_Example (* task: Scan Program *)
(* example of MC_SetPositionAll function block *)
VAR
    All_Axes_Ready : BOOL; (* flag that all axes are ready *)
    Execute_SetPositionAll : BOOL; (* execute MC_SetPositionAll function block *)
    SetPosition_Aborted : BOOL; (* aborted status for MC_SetPositionAll *)
    SetPosition_Busy : BOOL; (* busy status for MC_SetPositionAll *)
    SetPosition_Error : BOOL; (* error status for MC_SetPositionAll fb *)
    SetPosition_ErrorID : WORD; (* error identification for MC_SetPositionAll *)
    SetPosition_ExecutionMode : UINT; (* execution mode for MC_SetPositionAll *)
    SetPosition_INST : MC_SETPOSITIONALL; (* MC_SetPositionAll function block *)
    SetPosition_Position : LREAL; (* position to set to axes *)
    SetPosition_Relative : BOOL; (* 0 - Absolute Position change *)
END_VAR

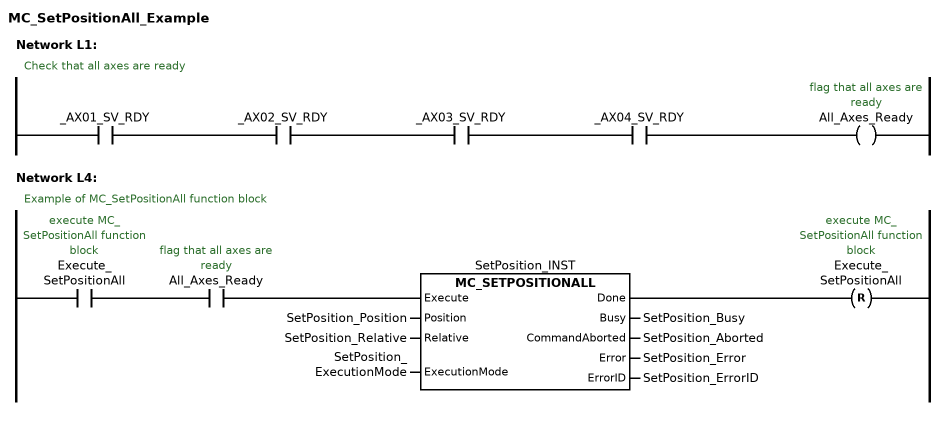
(* Check that all axes are ready *)
(* Rung L1 *)
All_Axes_Ready := _AX01_SV_RDY AND _AX02_SV_RDY AND _AX03_SV_RDY AND _AX04_SV_RDY;
(* Example of MC_SetPositionAll function block *)
(* Rung L4 *)
SetPosition_INST(Execute := Execute_SetPositionAll AND All_Axes_Ready, Position := SetPosition_Position, Relative := SetPosition_Relative, ExecutionMode := SetPosition_ExecutionMode, Busy => SetPosition_Busy, CommandAborted => SetPosition_Aborted, Error => SetPosition_Error, ErrorID => SetPosition_ErrorID);
IF SetPosition_INST.Done THEN Execute_SetPositionAll := FALSE; END_IF;
END_PROGRAM